(* CoDeSys 2.3.9.28 project: Aula12_furadeiraAutomatica.pro *)
(* Libraries: Standard.lib 27.1.09 11:27:38, Util.lib 27.1.09 11:27:38, IecSfc.lib 24.11.08 08:07:15, SysLibTime.lib 27.1.09 11:27:38, SysTaskInfo.lib 24.11.08 08:07:15, SYSLIBCALLBACK.LIB 27.1.09 11:27:38 *)

(* PLC configuration (modules and I/O channels)
CPX-CEC [Root] node -1, in %IB0 out %QB0 {StringParam = 2773,0,0,0,0; ByteParam = 0; ByteParam = 31; ByteParam = 0; ByteParam = 0; ByteParam = 0; ByteParam = 0; ByteParam = 0; ByteParam = 0; ByteParam = 2; ByteParam = 0; ByteParam = 0; ByteParam = 0; ByteParam = 32; ByteParam = 0; ByteParam = 0; ByteParam = 5; ByteParam = 0; ByteParam = 0; ByteParam = 0; ByteParam = 0; ByteParam = 0; ByteParam = 0; ByteParam = 0; ByteParam = 0; ByteParam = 14; ByteParam = 240; ByteParam = 192; ByteParam = 168; ByteParam = 2; ByteParam = 10; ByteParam = 255; ByteParam = 255; ByteParam = 0; ByteParam = 0; ByteParam = 192; ByteParam = 168; ByteParam = 1; ByteParam = 1; ByteParam = 192; ByteParam = 168; ByteParam = 2; ByteParam = 10; ByteParam = 255; ByteParam = 255; ByteParam = 0; ByteParam = 0; ByteParam = 192; ByteParam = 168; ByteParam = 1; ByteParam = 1}
  Hexswitch AT %IB0 [HexSwitch] rotary switch 0 = STOP, 1-15 = RUN
  IOModules [CPX_MASTER] node 0, in %IB4 out %QB0
*)

(* Global variable list: Global_Variables *)
VAR_GLOBAL

	START : BOOL;
	S1: BOOL;
	S2: BOOL;
	S3: BOOL;
	STOP: BOOL;

	C1 : BOOL;
	C2 : BOOL;
	M1 : BOOL;
	LAMP : BOOL;

	MEM1 : BOOL;

END_VAR

(* POU PLC_PRG, ST *)
PROGRAM PLC_PRG
VAR
END_VAR
IF START THEN
	LAMP := TRUE;
	C1 := TRUE;
	MEM1 := FALSE;
	M1 := FALSE;
	C2 := FALSE;

END_IF


IF S1 AND LAMP THEN
	M1 := TRUE;
	C2 := TRUE;

END_IF


IF S2 AND LAMP THEN
	MEM1 := TRUE;
	C2 := FALSE;

END_IF



IF (S3 AND MEM1) OR STOP THEN
	LAMP := FALSE;
	M1 := FALSE;
	C1 := FALSE;
	MEM1 := FALSE;
	C2 := FALSE;

END_IF
END_PROGRAM

(* Visualisation TELA
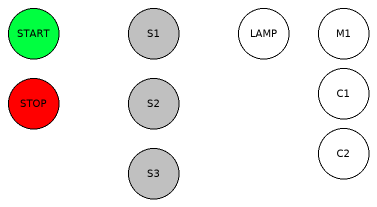
ellipse at (60,50)-(111,101): text "START"; alarm colour if START; taps START
ellipse at (60,120)-(111,171): text "STOP"; alarm colour if STOP; taps STOP
ellipse at (180,50)-(231,101): text "S1"; alarm colour if S1; taps S1
ellipse at (180,120)-(231,171): text "S2"; alarm colour if S2; taps S2
ellipse at (290,50)-(341,101): text "LAMP"; alarm colour if LAMP
ellipse at (370,110)-(421,161): text "C1"; alarm colour if C1
ellipse at (370,170)-(421,221): text "C2"; alarm colour if C2
ellipse at (180,190)-(231,241): text "S3"; alarm colour if S3; toggles S3
ellipse at (370,50)-(421,101): text "M1"; alarm colour if M1
*)
